// TIA Portal project "FactoryIO_Template_S7-1200_V15_V16" (V16)
// Vorlageprojekt für das Buch mit Zielsystem S7-1200

(* hardware
DEVICE "S7-1200-Station_1"  S7-1200 Station
   slot 0: "Baugruppenträger_0"  Rack  V1.0
   slot 1: "PLC_1"  CPU 1211C DC/DC/DC  6ES7 211-1AE40-0XB0  V4.1
*)

// ===== PLC "PLC_1"  CPU 1211C DC/DC/DC =====

VAR_GLOBAL   // PLC tag table "Standard-Variablentabelle"
   "Start" AT %I0.0 : Bool;
   "Stop" AT %I0.1 : Bool;
   "Base Detector" AT %I0.2 : Bool;
   "Base Clamped" AT %I0.3 : Bool;
   "Base Clamp Raised" AT %I0.4 : Bool;
   "Lid Detector" AT %I0.5 : Bool;
   "Lid Clamped" AT %I0.6 : Bool;
   "Gripper Moving X" AT %I0.7 : Bool;
   "Gripper Moving Z" AT %I1.0 : Bool;
   "Gripper-Touched lid" AT %I1.1 : Bool;
   "Product Detector" AT %I1.2 : Bool;
   "Collection Box Limit" AT %I1.3 : Bool;
   "Turnable Back Limit" AT %I1.4 : Bool;
   "Turnable Front Limit" AT %I1.5 : Bool;
   "Turnable Limit 90" AT %I1.7 : Bool;
   "Base Material emitter" AT %Q0.0 : Bool;
   "Lid Material Emitter" AT %Q0.1 : Bool;
   "Base Clamp" AT %Q0.2 : Bool;
   "Lid Output Conveyor" AT %Q0.3 : Bool;
   "base Clamp Raise" AT %Q0.4 : Bool;
   "Lid Clamp" AT %Q0.5 : Bool;
   "Bottle Output Conveyor" AT %Q0.6 : Bool;
   "Product Output Conveyor" AT %Q0.7 : Bool;
   "Collection Box emitter" AT %Q1.0 : Bool;
   "Gripper-Move X" AT %Q1.1 : Bool;
   "Gripper-Move Z" AT %Q1.2 : Bool;
   "Gripper-Grab" AT %Q1.3 : Bool;
   "Turntable Roll(+)" AT %Q1.4 : Bool;
   "Turntable Turn" AT %Q1.5 : Bool;
   "Turntable Roll(-)" AT %Q1.6 : Bool;
   "Base Aligned" AT %M0.1 : Bool;
   "Lid Aligned" AT %M0.2 : Bool;
   "Lid Grabbed" AT %M0.3 : Bool;
   "Lid Above 'Lid Clamp'" AT %M0.4 : Bool;
   "Lid Above Base" AT %M0.5 : Bool;
   "Product Assembled" AT %M0.6 : Bool;
END_VAR

// folder: System blocks/Program resources

DATA_BLOCK "IEC_Timer_0_DB"   // DB1
{ S7_Optimized_Access := 'TRUE' }
AUTHOR : Simatic
FAMILY : IEC
NAME : IEC_TMR
VERSION : 1.0
// stored: InstanceOfName IEC_TIMER
"IEC_TIMER"
BEGIN
END_DATA_BLOCK

DATA_BLOCK "IEC_Timer_0_DB_1"   // DB2
{ S7_Optimized_Access := 'TRUE' }
AUTHOR : Simatic
FAMILY : IEC
NAME : IEC_TMR
VERSION : 1.0
// stored: InstanceOfName IEC_TIMER
"IEC_TIMER"
BEGIN
END_DATA_BLOCK

DATA_BLOCK "IEC_Timer_0_DB_2"   // DB3
{ S7_Optimized_Access := 'TRUE' }
AUTHOR : Simatic
FAMILY : IEC
NAME : IEC_TMR
VERSION : 1.0
// stored: InstanceOfName IEC_TIMER
"IEC_TIMER"
BEGIN
END_DATA_BLOCK

DATA_BLOCK "IEC_Timer_0_DB_3"   // DB4
{ S7_Optimized_Access := 'TRUE' }
AUTHOR : Simatic
FAMILY : IEC
NAME : IEC_TMR
VERSION : 1.0
// stored: InstanceOfName IEC_TIMER
"IEC_TIMER"
BEGIN
END_DATA_BLOCK

DATA_BLOCK "IEC_Timer_0_DB_4"   // DB5
{ S7_Optimized_Access := 'TRUE' }
AUTHOR : Simatic
FAMILY : IEC
NAME : IEC_TMR
VERSION : 1.0
// stored: InstanceOfName IEC_TIMER
"IEC_TIMER"
BEGIN
END_DATA_BLOCK

DATA_BLOCK "IEC_Timer_0_DB_5"   // DB6
{ S7_Optimized_Access := 'TRUE' }
AUTHOR : Simatic
FAMILY : IEC
NAME : IEC_TMR
VERSION : 1.0
// stored: InstanceOfName IEC_TIMER
"IEC_TIMER"
BEGIN
END_DATA_BLOCK

DATA_BLOCK "IEC_Timer_0_DB_6"   // DB7
{ S7_Optimized_Access := 'TRUE' }
AUTHOR : Simatic
FAMILY : IEC
NAME : IEC_TMR
VERSION : 1.0
// stored: InstanceOfName IEC_TIMER
"IEC_TIMER"
BEGIN
END_DATA_BLOCK

DATA_BLOCK "IEC_Timer_0_DB_7"   // DB8
{ S7_Optimized_Access := 'TRUE' }
AUTHOR : Simatic
FAMILY : IEC
NAME : IEC_TMR
VERSION : 1.0
// stored: InstanceOfName IEC_TIMER
"IEC_TIMER"
BEGIN
END_DATA_BLOCK

DATA_BLOCK "IEC_Timer_0_DB_8"   // DB9
{ S7_Optimized_Access := 'TRUE' }
AUTHOR : Simatic
FAMILY : IEC
NAME : IEC_TMR
VERSION : 1.0
// stored: InstanceOfName IEC_TIMER
"IEC_TIMER"
BEGIN
END_DATA_BLOCK

DATA_BLOCK "IEC_Timer_0_DB_9"   // DB10
{ S7_Optimized_Access := 'TRUE' }
AUTHOR : Simatic
FAMILY : IEC
NAME : IEC_TMR
VERSION : 1.0
// stored: InstanceOfName IEC_TIMER
"IEC_TIMER"
BEGIN
END_DATA_BLOCK

// folder: (top level)

FUNCTION "MHJ-PLC-Lab-Function-S71200" : Void   // FC9000, SCL
{ S7_Optimized_Access := 'TRUE' }
VERSION : 0.1
   VAR_TEMP
      rdTimeReturn : Int;
      outputTime : DTL;
      SyncVal : Byte;
      forVal : Int;
      forVal_2 : Int;
      Value : Byte;
   END_VAR
   VAR CONSTANT
      CompVal : Byte := 16#34;
      Value_01 : Byte := 16#11;
      Value_01_DW : DWord := 16#A165_D992;
      Value_02_DW : DWord := 16#58BE_4401;
   END_VAR
BEGIN

   #Value:=PEEK(area := 16#82,
        dbNumber := 0,
        byteOffset := 511);
   #Value := #Value + 1;

   POKE(area := 16#82,
        dbNumber := 0,
        byteOffset := 511,
        value := #Value);

   POKE(area:=16#81,
        dbNumber:=0,
        byteOffset:=1016,
        value:=#Value_01_DW);
   POKE(area := 16#81,
        dbNumber := 0,
        byteOffset := 1020,
        value := #Value_02_DW);

   POKE(area := 16#81,
        dbNumber := 0,
        byteOffset := 511,
        value := B#16#00);

   FOR #forVal := 0 TO 120 DO
       FOR #forVal_2:=0 TO 10 DO
           #rdTimeReturn:=RD_SYS_T(#outputTime);
           #rdTimeReturn := WR_SYS_T(#outputTime);
           #rdTimeReturn := RD_SYS_T(#outputTime);
           #rdTimeReturn := WR_SYS_T(#outputTime);
       END_FOR;
       #SyncVal:= PEEK(area := 16#81,
                      dbNumber := 0,
                      byteOffset := 511);
       IF #SyncVal = #CompVal THEN
          GOTO M_1;
       END_IF;
   END_FOR;
   RETURN;

   M_1:
   POKE(area := 16#81,
        dbNumber := 0,
        byteOffset := 511,
        value := B#16#0);
END_FUNCTION

ORGANIZATION_BLOCK "Main"   // OB1, LAD, ProgramCycle
TITLE = "Main Program Sweep (Cycle)"
{ S7_Optimized_Access := 'TRUE' }
VERSION : 0.1
   VAR_INPUT
      Initial_Call : Bool;   // Initial call of this OB
      Remanence : Bool;   // =True, if remanent data are available
   END_VAR
   VAR_TEMP   // added for the SCL form of the ladder/FBD networks
      _w1 : Bool;
   END_VAR
BEGIN

REGION Network 1: Konnektierungsbaustein für PLC-Lab
   // Im Netzwerk 1 wird der Konnektierungsbaustein für PLC-Lab aufgerufen.
   // Dieser Aufruf darf nicht entfernt werden!
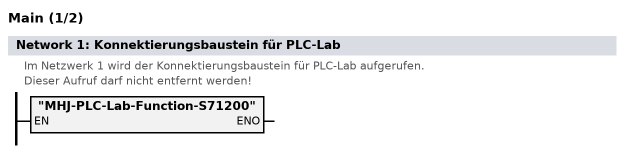
   RUNG wire#powerrail
      "MHJ-PLC-Lab-Function-S71200"()
   END_RUNG
   // the same network as SCL:
   "MHJ-PLC-Lab-Function-S71200"();
END_REGION

REGION Network 2: Ihr Programm
   // Schreiben Sie ab Netzwerk 2 Ihr Programm
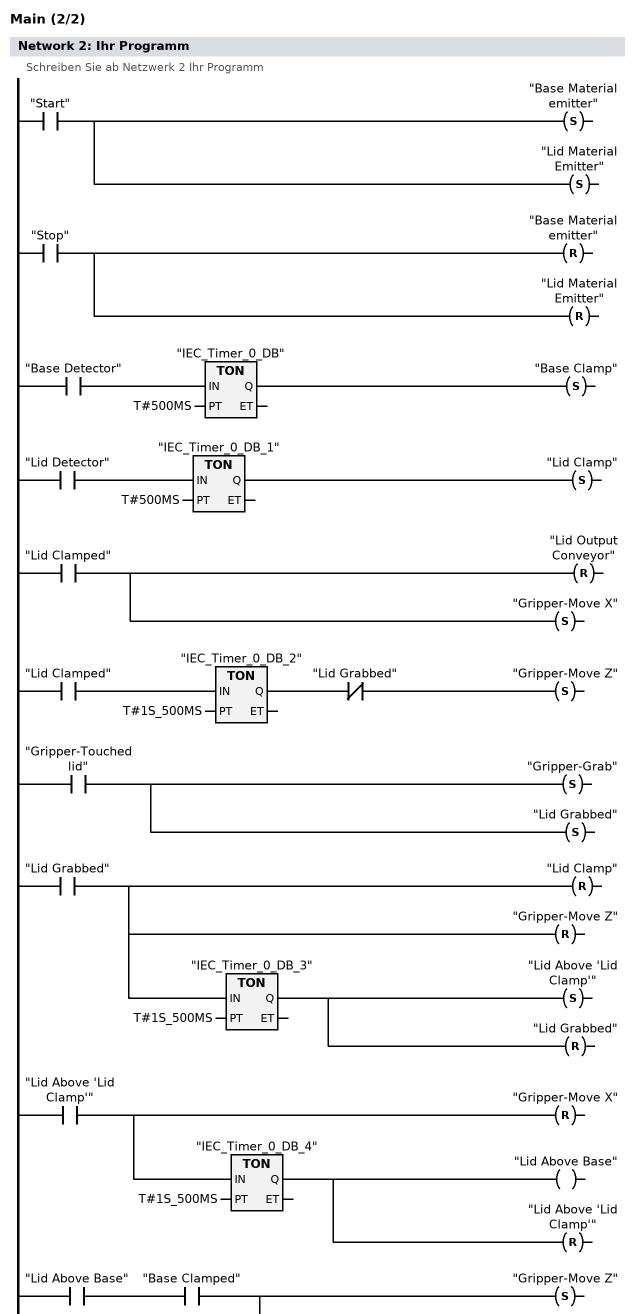
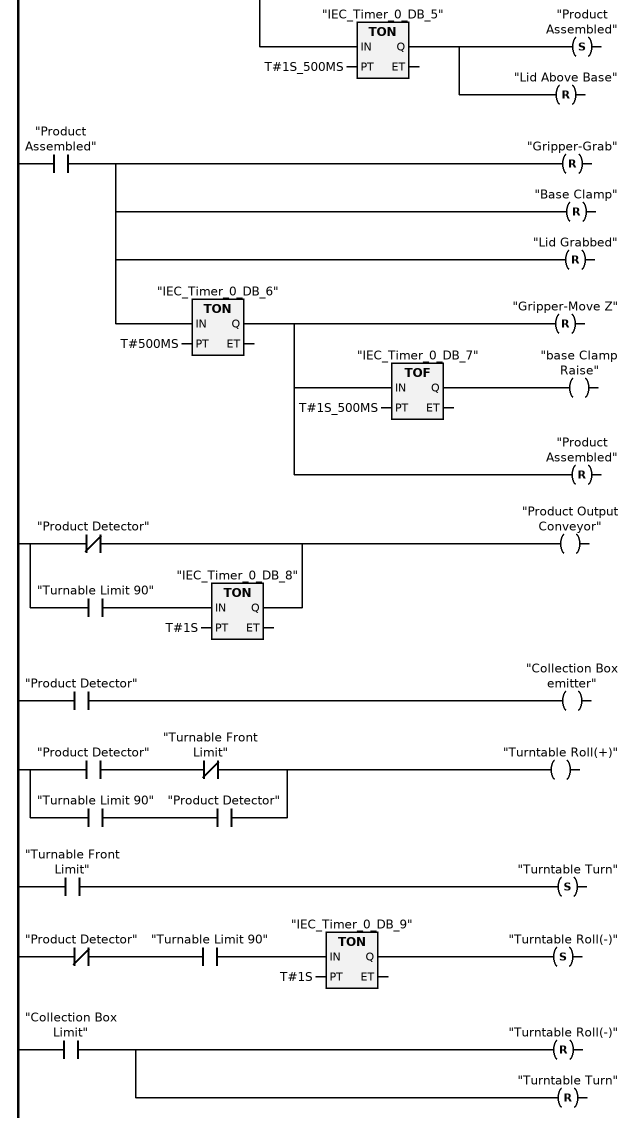
   IF "Start" THEN
       "Base Material emitter" := TRUE;
       "Lid Material Emitter" := TRUE;
   END_IF;
   IF "Stop" THEN
       "Base Material emitter" := FALSE;
       "Lid Material Emitter" := FALSE;
   END_IF;
   "IEC_Timer_0_DB".TON(IN := "Base Detector", PT := T#500MS);
   IF "IEC_Timer_0_DB".Q THEN "Base Clamp" := TRUE; END_IF;
   "IEC_Timer_0_DB_1".TON(IN := "Lid Detector", PT := T#500MS);
   IF "IEC_Timer_0_DB_1".Q THEN "Lid Clamp" := TRUE; END_IF;
   IF "Lid Clamped" THEN
       "Lid Output Conveyor" := FALSE;
       "Gripper-Move X" := TRUE;
   END_IF;
   "IEC_Timer_0_DB_2".TON(IN := "Lid Clamped", PT := T#1S_500MS);
   IF "IEC_Timer_0_DB_2".Q AND NOT "Lid Grabbed" THEN "Gripper-Move Z" := TRUE; END_IF;
   IF "Gripper-Touched lid" THEN
       "Gripper-Grab" := TRUE;
       "Lid Grabbed" := TRUE;
   END_IF;
   IF "Lid Grabbed" THEN
       "Lid Clamp" := FALSE;
       "Gripper-Move Z" := FALSE;
   END_IF;
   "IEC_Timer_0_DB_3".TON(IN := "Lid Grabbed", PT := T#1S_500MS);
   IF "IEC_Timer_0_DB_3".Q THEN
       "Lid Above 'Lid Clamp'" := TRUE;
       "Lid Grabbed" := FALSE;
   END_IF;
   IF "Lid Above 'Lid Clamp'" THEN "Gripper-Move X" := FALSE; END_IF;
   "IEC_Timer_0_DB_4".TON(IN := "Lid Above 'Lid Clamp'", PT := T#1S_500MS);
   "Lid Above Base" := "IEC_Timer_0_DB_4".Q;
   IF "IEC_Timer_0_DB_4".Q THEN "Lid Above 'Lid Clamp'" := FALSE; END_IF;
   #_w1 := "Lid Above Base" AND "Base Clamped";
   IF #_w1 THEN "Gripper-Move Z" := TRUE; END_IF;
   "IEC_Timer_0_DB_5".TON(IN := #_w1, PT := T#1S_500MS);
   IF "IEC_Timer_0_DB_5".Q THEN
       "Product Assembled" := TRUE;
       "Lid Above Base" := FALSE;
   END_IF;
   IF "Product Assembled" THEN
       "Gripper-Grab" := FALSE;
       "Base Clamp" := FALSE;
       "Lid Grabbed" := FALSE;
   END_IF;
   "IEC_Timer_0_DB_6".TON(IN := "Product Assembled", PT := T#500MS);
   IF "IEC_Timer_0_DB_6".Q THEN "Gripper-Move Z" := FALSE; END_IF;
   "IEC_Timer_0_DB_7".TOF(IN := "IEC_Timer_0_DB_6".Q, PT := T#1S_500MS);
   "base Clamp Raise" := "IEC_Timer_0_DB_7".Q;
   IF "IEC_Timer_0_DB_6".Q THEN "Product Assembled" := FALSE; END_IF;
   "IEC_Timer_0_DB_8".TON(IN := "Turnable Limit 90", PT := T#1S);
   "Product Output Conveyor" := NOT "Product Detector" OR "IEC_Timer_0_DB_8".Q;
   "Collection Box emitter" := "Product Detector";
   "Turntable Roll(+)" := ("Product Detector" AND NOT "Turnable Front Limit") OR ("Turnable Limit 90" AND "Product Detector");
   IF "Turnable Front Limit" THEN "Turntable Turn" := TRUE; END_IF;
   "IEC_Timer_0_DB_9".TON(IN := NOT "Product Detector" AND "Turnable Limit 90", PT := T#1S);
   IF "IEC_Timer_0_DB_9".Q THEN "Turntable Roll(-)" := TRUE; END_IF;
   IF "Collection Box Limit" THEN
       "Turntable Roll(-)" := FALSE;
       "Turntable Turn" := FALSE;
   END_IF;
END_REGION
END_ORGANIZATION_BLOCK